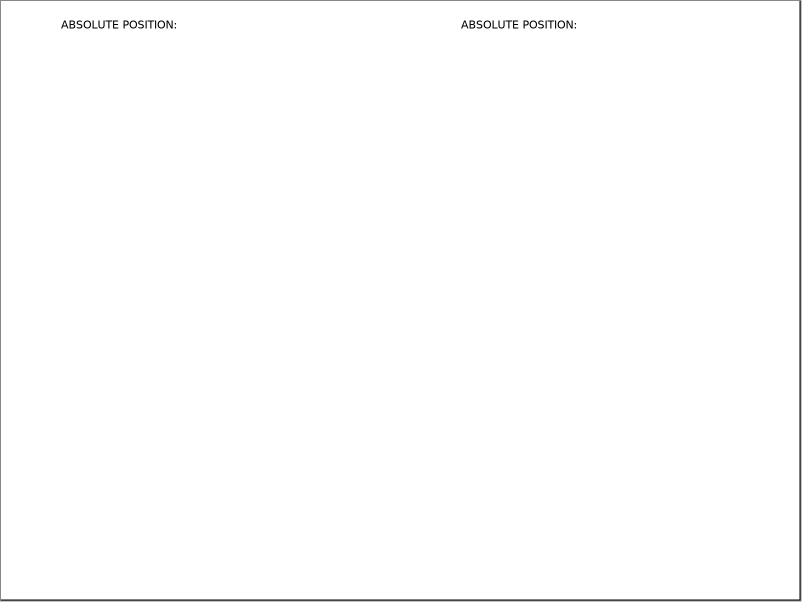
VISUALIZATION F35_Move_Modulo  // 802x602
    Rectangle (0,0 800x600)
    Label (10,10 170x30), "ABSOLUTE POSITION:"
    Label (410,10 170x30), "ABSOLUTE POSITION:"
END_VISUALIZATION

(* stored: Version 1.1.0.1, ProductVersion 3.1.4022.7
   Visu F35_Move_Modulo: Id {269e93d4-1863-4c78-b07c-913f74da1238} *)
